FUNCTION_BLOCK GearMover EXTENDS FB_Mover IMPLEMENTS IGearMover
VAR_INPUT
	StateMachine : IPmlStateMachine;
END_VAR
VAR_OUTPUT
END_VAR
VAR
	moverSequence : GearMoverSequence;
	bInit : BOOL;
	CurrentLimit AT%Q* : INT;
	Mode AT%Q* : UINT;
	axesGear	: GearInCA;
	isMasterAxis: BOOL;
	MoverToGearTo: UDINT := 1;
END_VAR
VAR_IN_OUT
	MoverArray : ARRAY[*] OF IGearMover;
END_VAR

METHOD PUBLIC  Cycle : BOOL
VAR_INPUT
END_VAR
IF NOT bInit THEN
	IF THIS^._axis.NcToPlc.AxisId <> 0 THEN
		IF (THIS^._axis.NcToPlc.AxisId MOD 2)<>1 THEN
			Mode.8 := TRUE;
			isMasterAxis := TRUE;
		ELSE
			isMasterAxis := FALSE;
			MoverToGearTo := THIS^.AxisRef.NcToPlc.AxisId + 1;
		END_IF
		bInit := TRUE;
	END_IF
END_IF

IF isMasterAxis THEN
	IF (_axis.NcToPlc.ModuloActPos > 3400 OR _axis.NcToPlc.ModuloActPos < 300)  THEN
		CurrentLimit := 1000;
	ELSE
		CurrentLimit := 2000;
	END_IF
ELSE
	CurrentLimit := 12000;
END_IF

SUPER^.Cycle();
axesGear(_MasterAxis := MoverArray[MoverToGearTo].AxisRef, _SlaveAxis := THIS^.AxisRef);
moverSequence(ThisMover := THIS^,
				StateMachine := StateMachine,
				MoverArray := MoverArray);
END_METHOD

METHOD PUBLIC Gear : BOOL
VAR_INPUT
	MasterPosition : MC_LREAL;
	SlavePosition : MC_LREAL;
END_VAR
IF NOT axesGear.Busy THEN
		Gear := axesGear.Sync(MasterPosition := MasterPosition, SlavePosition := SlavePosition);
END_IF
END_METHOD

METHOD inGear : BOOL
VAR_INPUT
END_VAR
inGear := axesGear.gearInCA.InSync;
END_METHOD

METHOD isMaster : BOOL
VAR_INPUT
END_VAR
isMaster := isMasterAxis;
END_METHOD

METHOD masterAxis : UDINT
VAR_INPUT
END_VAR
masterAxis := MoverToGearTo;
END_METHOD

END_FUNCTION_BLOCK

(* stored: Version 1.1.0.1, ProductVersion 3.1.4024.12
   POU GearMover: Id {e1672d47-cce7-4d2e-b6b6-6b7bf615c986}, SpecialFunc None
   Method Cycle: Id {675a77a0-454d-47dc-a1a2-22dd4fd08b5c}
   Method Gear: Id {b0aa32af-e1ad-43df-b90e-7e7d830bc963}
   Method inGear: Id {0809336a-3200-4d64-8806-8b040d87d191}
   Method isMaster: Id {f7cde0d7-54e3-403f-8a16-457e977c3959}
   Method masterAxis: Id {90bc7a08-10e6-4dcc-996f-38b71e0675dc} *)
